// TIA Portal V20 export
TYPE "UDT_MTP_MonBinVlv"
TITLE = MTPDataObjectSUCLibrary/DataAssembly/BinVlv
   STRUCT
      CloseOp : Bool := FALSE;   // Close command from Operator (relevant, if StateOpAct) 0-->1:request from POL 1-->0 acknowledge from PEA(see Handshake)
      OpenOp : Bool := FALSE;   // Open command from Operator (relevant, if StateOpAct) 0-->1:request from POL 1-->0 acknowledge from PEA(see Handshake)
      OSLevel : Byte := 16#00;   // OSLevel variable
      StateChannel { ExternalWritable := 'False'} : Bool;   // Selection of the active OperationMode interaction channel0: The operator switches (*Op) shall be used.1: The automatic switches (*Aut) shall be used.
      StateOffAut { ExternalWritable := 'False'} : Bool;   // Set OperationMode to Offline by automatic interaction (relevant, if StateChannel).1: OperationMode is set to Offline.0: no operation
      StateOffOp : Bool;   // Set OperationMode to Offline by operator interaction (relevant, if not StateChannel) 0-->1:request to set OperationMode to Offline 1-->0:acknowledge by PEA
      StateOpAut { ExternalWritable := 'False'} : Bool;   // Set OperationMode to Operator by automatic interaction (relevant, if StateChannel).1: OperationMode is set to Manual.0: no operation
      StateOpOp : Bool;   // Set OperationMode to Offline by operator interaction (relevant, if not StateChannel) 0-->1:request to set OperationMode to Offline 1-->0:acknowledge by PEA
      StateAutAut { ExternalWritable := 'False'} : Bool;   // Set OperationMode to Automatic by automatic interaction (relevant, if StateChannel).1: OperationMode is set to Automatic.0: no operation
      StateAutOp : Bool;   // Set OperationMode to Automatic by operator interaction (relevant, if not StateChannel) 0-->1:request to set OperationMode is to Automatic 1-->0:acknowledge by PEA
      StateOpAct { ExternalWritable := 'False'} : Bool;   // 1: current mode is Operator0: current mode is not Operator
      StateAutAct { ExternalWritable := 'False'} : Bool;   // 1: current mode is Automatic0: current mode is not Automatic
      StateOffAct { ExternalWritable := 'False'} : Bool;   // 1: current mode is Offline0: current mode is not Offline
      CSF { ExternalWritable := 'False'} : Bool;   // Reserved
      WQC { ExternalWritable := 'False'} : Byte := 16#FF;   // Worst Quality Code variable
      CloseAut { ExternalWritable := 'False'} : Bool := FALSE;   // Set Valve to Close by Automatic.(relevant, if StateAutAct)1: close request0: no close request
      OpenAut { ExternalWritable := 'False'} : Bool := FALSE;   // Set Valve to Open by Automatic.(relevant, if StateAutAct)1: open request0: no open request
      Ctrl { ExternalWritable := 'False'} : Bool := FALSE;   // Valve Control1: desired position is open0: desired position is closed
      OpenFbkCalc { ExternalWritable := 'False'} : Bool := FALSE;   // Open Feedback Source1: calculated0: sensor detection
      CloseFbkCalc { ExternalWritable := 'False'} : Bool := FALSE;   // Close Feedback Source1: Calculated0: Sensor detection
      OpenFbk { ExternalWritable := 'False'} : Bool := FALSE;   // Open Feedback Signal1: open0: is not opened
      CloseFbk { ExternalWritable := 'False'} : Bool := FALSE;   // Close Feedback Signal1: Close0: is not closed
      SafePos { ExternalWritable := 'False'} : Bool := FALSE;   // Safe Position1: open0: close
      SafePosEn { ExternalWritable := 'False'} : Bool;   // Hardware Safe Position enabled1: Device has a safe position.0: Device has no safe position.
      SafePosAct { ExternalWritable := 'False'} : Bool;   // Safe Position activated 1: Safe Position is activated (safe operation) 0: Safe Position is not activated (normal operation)
      PermEn { ExternalWritable := 'False'} : Bool := FALSE;   // Enables the Permission Lock1: enabled0: disabled
      Permit { ExternalWritable := 'False'} : Bool := FALSE;   // Permit allows control1: permission is given0: permission is not given
      IntlEn { ExternalWritable := 'False'} : Bool := FALSE;   // Enables the Interlock Lock1: enabled0: disabled
      Interlock { ExternalWritable := 'False'} : Bool := FALSE;   // Interlock prevents from being activated and sets it to safe position.1: Interlock is not active0: Interlock is active
      ProtEn { ExternalWritable := 'False'} : Bool := FALSE;   // Enables the Protection Lock1: enabled; 0: disabled
      Protect { ExternalWritable := 'False'} : Bool := FALSE;   // Protect prevents from being activated and sets it to safe position, requires a reset command.1: protect is not active0: protect is active, requires reset
      ResetOp : Bool := FALSE;   // Reset from Operator (see Handshake) 0-->1:request from POL 1-->0: acknowledge from PEA
      ResetAut { ExternalWritable := 'False'} : Bool;   // Reset from Automatic1: Reset execute0: no operation
      MonEn : Bool := FALSE;   // Monitor Enable1: enabled0: disabled
      MonSafePos { ExternalWritable := 'False'} : Bool := FALSE;   // Set the Error Behavior, if an error occurs.1: After an error occurs, the Safe Position will be set.0: After an error occurs, the entity holds the state.
      MonStatErr { ExternalWritable := 'False'} : Bool := FALSE;   // Static Error active1: active0: inactive
      MonDynErr { ExternalWritable := 'False'} : Bool := FALSE;   // Dynamic Error active1: active0: inactive
      MonStatTi { ExternalWritable := 'False'} : Real := 0.0;   // Monitor Time for uncontrolled changes, in s
      MonDynTi { ExternalWritable := 'False'} : Real := 0.0;   // Monitor Time for controlled changes, in s
   END_STRUCT;
END_TYPE
